// TIA Portal V19 export
VAR_GLOBAL   // PLC tag table "MES_MSG_KEYS_CONST"
END_VAR
VAR_GLOBAL CONSTANT   // user constants
   MES_MSG_KEY_SEPARATOR : String := ';';   // separatore coppia chiave valore
   MES_MSG_IDP : String := '[IDP]=';   // Identificativo univoco che indentifica l’ordine di produzione sul lato PLC
   MES_MSG_TYP : String := '[TYP]=';   // Tipo profilo (es. S, C)
   MES_MSG_W : String := '[W]=';   // Base del pezzo (es. 40)
   MES_MSG_H : String := '[H]=';   // Altezza del pezzo (es. 60)
   MES_MSG_TK : String := '[TK]=';   // Spessore (es. 1.25)
   MES_MSG_LN : String := '[LN]=';   // Lunghezza del pezzo in mm
   MES_MSG_QQ : String := '[QQ]=';   // Quantità di pezzi da eseguire
   MES_MSG_RR : String := '[RR]=';   // Profilo nervato (No=0; Si=>=1)
   MES_MSG_DC : String := '[DC]=';   // Uso marchio identificazione tracciabilità (colata?) (No=0; Si=>=1)
   MES_MSG_DE : String := '[DE]=';   // Uso marchio identificazione MODULBLOK (No=0; Si=>=1)
   MES_MSG_KA : String := '[KA]=';   // Stile Kanban (No=0; Si=>=1).*1
   MES_MSG_NPR : String := '[NPR]=';   // Schema pallettizzazione: Numero pezzi per strati.
   MES_MSG_NPL : String := '[NPL]=';   // Schema palettizzazione: Numero strati.
   MES_MSG_IDI : String := '[IDI]=';   // ID messaggio di interrogazione
   MES_MSG_SOR : String := '[SOR]=';   // Stato ordine di produzione
   MES_MSG_STSP : String := '[STSP]=';   // Stato sospensione produzione semi-gusci
   MES_MSG_STS : String := '[STS]=';   // Stato sospensione produzione pezzi finiti
   MES_MSG_QG : String := '[QG]=';   // Numero pezzi conformi
   MES_MSG_QGR : String := '[QGR]=';   // Pezzi conformi dopo ricondizionamento
   MES_MSG_QNG : String := '[QNG]=';   // Numero pezzi non conformi
   MES_MSG_QPG : String := '[QPG]=';   // Numero semi-gusci conformi
   MES_MSG_QPGR : String := '[QPGR]=';   // Semi-gusci conformi dopo ricondizionamento
   MES_MSG_QPNG : String := '[QPNG]=';   // Semi-gusci non conformi
   MES_MSG_SPP : String := '[SPP]=';   // Stato pacco baia preparazione
   MES_MSG_QTY : String := '[QTY]=';   // Quantità richiesta pacco
   MES_MSG_QPR : String := '[QPR]=';   // Pezzi nello strato incompleto
   MES_MSG_QPL : String := '[QPL]=';   // Strati completati
   MES_MSG_SPU : String := '[SPU]=';   // Stato pacco baia uscita
   MES_MSG_DT : String := '[DT]=';   // Timestamp evento
   MES_MSG_IC : String := '[IC]=';   // Codice causa sospensione
   MES_MSG_MC : String := '[MC]=';   // Codice allarme/warning
   MES_MSG_CN : String := '[CN]=';   // Numero identificativo rotolo
   MES_MSG_HN : String := '[HN]=';   // Numero colata
   MES_MSG_PR : String := '[PR]=';   // Richiesta provino
   MES_MSG_SR : String := '[SR]=';   // Stato rotolo
   MES_MSG_PRR : String := '[PRR]=';   // Numero provini richiesti
   MES_MSG_PRD : String := '[PRD]=';   // Numero provini eseguiti
   MES_MSG_TNG : String := '[TNG]=';   // Errore spessore rilevato
   MES_MSG_TKD : String := '[TKD]=';   // Uso rotolo in deroga
   MES_MSG_SL : String := '[SL]=';   // Lunghezza materiale scartato
   MES_MSG_SC : String := '[SC]=';   // Codice causa scarto
   MES_MSG_TEV : String := '[TEV]=';   // Valore dello spessore fuori tolleranza
   MES_MSG_RDM : String := '[RDM]=';   // Diametro del rotolo
   MES_MSG_TAV : String := '[TAV]=';   // Valore dello spessore letto dal sensore
END_VAR
